FUNCTION_BLOCK FB_Regelschuif_AFO IMPLEMENTS ITF_Regelschuif
VAR
	tagName : STRING;
	outputOpen : ITF_Schuif_DigOutOpen_AFO;
	outputClose : ITF_Schuif_DigOutClose_AFO;
	inputPosition : ITF_Schuif_AnaIn_AFO;

	currentMode : E_Bedrijfstoestand := E_Bedrijfstoestand.off;
	currentState : E_RegelschuifState := E_RegelschuifState.standby;
	expectedState : E_RegelschuifState := E_RegelschuifState.standby;
	
	feedbackPosition : SINT;
	
	timeOut : TON;
	errorTrigger : R_TRIG;
	positie : SINT;
	secondTimerRun : BOOL;
	secondTimerTrigger : R_TRIG;
	
	timerrunt: BOOL:=1;
	waitExtraMinute: BOOL;
	minuteTimer : TON;
	doubleMinuteTimer : TON;
	secondTimer : TON;
	
	veranderingsMargeError : SINT := 3;
	OldPosition: SINT;
	regelschuifMargin: SINT := 3;
END_VAR

// Als de mode is uit dan worden de outputs false geset 
IF currentMode = E_Bedrijfstoestand.off THEN
	outputOpen.set(FALSE);
	outputClose.set(FALSE);
END_IF

// De feedback positie staat hiet zodat we de waardes kunnen veranderen
feedbackPosition := inputPosition.get();
ActueelPosition := inputPosition.get();

// Dit is de timer om te checken of er een error moet zijn 
timeOut(IN :=(StateRegelSchuif <> E_RegelschuifState.standby) AND NOT timeOut.Q, PT := T#30S);
errorTrigger(CLK := timeOut.Q);

IF errorTrigger.Q THEN
	IF (ActueelPosition < (OldPosition + veranderingsMargeError)) AND StateRegelSchuif = E_RegelschuifState.opening THEN
		StateRegelSchuif := E_RegelschuifState.error;
		main.alarms.append(tag := tagName, msg := 'Schuifstoring gedetecteerd, te langzaam openen');
	END_IF
	IF (ActueelPosition > (OldPosition - veranderingsMargeError)) AND StateRegelSchuif = E_RegelschuifState.closing THEN
		StateRegelSchuif := E_RegelschuifState.error;
		main.alarms.append(tag := tagName, msg := 'Schuifstoring gedetecteerd, te langzaam sluiten');
	END_IF
	IF StateRegelSchuif = E_RegelschuifState.error AND (ActueelPosition > (OldPosition + veranderingsMargeError)) THEN
		StateRegelSchuif := E_RegelschuifState.opening;
		ELSIF StateRegelSchuif = E_RegelschuifState.error AND (ActueelPosition < (OldPosition - veranderingsMargeError)) THEN
			StateRegelSchuif := E_RegelschuifState.closing;
	END_IF
	OldPosition := ActueelPosition;
END_IF

expectedState := StateRegelSchuif;

PROPERTY ActueelPosition : SINT
GET
ActueelPosition := feedbackPosition;
END_GET
SET
feedbackPosition := ActueelPosition;
END_SET
END_PROPERTY

//FB_Init is always available implicitly and it is used primarily for initialization.
//The return value is not evaluated. For a specific influence, you can also declare the
//methods explicitly and provide additional code there with the standard initialization
//code. You can evaluate the return value.
METHOD FB_Init: BOOL
VAR_INPUT
    bInitRetains: BOOL; // TRUE: the retain variables are initialized (reset warm / reset cold)
    bInCopyCode: BOOL;  // TRUE: the instance will be copied to the copy code afterward (online change)   
	tag : STRING;
	DigOutOpening : ITF_Schuif_DigOutOpen_AFO;
	DigOutClosing : ITF_Schuif_DigOutClose_AFO;
	AnaInPosition : ITF_Schuif_AnaIn_AFO;
END_VAR
tagname := tag;
outputOpen := DigOutOpening;
outputClose := DigOutClosing;
inputPosition := AnaInPosition;
END_METHOD

METHOD RegelSchuifGoTo : SINT
VAR	
	checkPositions : BOOL;
	currentstatet: E_RegelschuifState;
	secondTriggerTrigger: BOOL;
END_VAR
VAR_INPUT
	regelschuifdoel : SINT;
END_VAR
minuteTimer(IN:= timerrunt,PT:= T#10S);
doubleMinuteTimer(IN:= waitExtraMinute,PT:= T#10S); // tweede timer om een extra minuut te wachten na pulse maar niet langer te wachten met scannen

// dit is zodat het gefaseerd gaat een pulse per sec sturen
secondTimer(IN:= secondTimerRun,PT:= T#2S); // pulse lengte langer ivm testen

IF currentMode = E_Bedrijfstoestand.off THEN
	regelschuifdoel := ActueelPosition;
END_IF

IF minuteTimer.Q THEN
	
	IF ActueelPosition >= (regelschuifdoel - regelschuifMargin) AND ActueelPosition <= (regelschuifdoel + regelschuifMargin) THEN // huidige positie is correct binnen marge
		StateRegelSchuif := E_RegelschuifState.standby;
		outputOpen.set(FALSE); // set outputs naar 0 als extra backup
		outputClose.set(FALSE);
	
	END_IF
	
	IF ActueelPosition > (regelschuifdoel + regelschuifMargin) AND waitExtraMinute = FALSE THEN // huidige positie is te hoog
		IF stateRegelschuif <> E_RegelschuifState.error THEN
			StateRegelSchuif := E_RegelschuifState.closing;
		END_IF
		// voor de pulse		
		outputOpen.set(FALSE);
		outputClose.set(TRUE);
		secondTimerRun := TRUE; // start pulse time
		waitExtraMinute := TRUE; // wacht een minuut extra als er een pulse is gestuurd
	END_IF

	IF ActueelPosition < (regelschuifdoel - regelschuifMargin) AND waitExtraMinute = FALSE THEN // huidige positie is te laag
		IF stateRegelschuif <> E_RegelschuifState.error THEN
			StateRegelSchuif := E_RegelschuifState.opening;
		END_IF
		// voor de pulse
		outputClose.set(FALSE);
		outputOpen.set(TRUE);
		secondTimerRun := TRUE; // start pulse time
		waitExtraMinute := TRUE;
	END_IF
	timerrunt := 0; // reset timer
ELSIF waitExtraMinute = FALSE OR doubleMinuteTimer.Q THEN 
	waitExtraMinute := FALSE;
	timerrunt := 1; //reser reset timer
END_IF

// pulse timer structuur
IF secondTimer.Q THEN
	outputClose.set(FALSE);
	outputOpen.set(FALSE);
	secondTimerRun := FALSE;
END_IF

positie := regelschuifdoel;
END_METHOD

PROPERTY StateRegelSchuif : E_RegelschuifState
GET
StateRegelschuif := currentState;
END_GET
SET
currentstate:= StateRegelSchuif;
END_SET
END_PROPERTY

END_FUNCTION_BLOCK

(* stored: Version 1.1.0.1, ProductVersion 3.1.4026.8
   POU FB_Regelschuif_AFO: Id {e3716e21-c926-4b53-b092-edc4b4bb1690}, SpecialFunc None
   Folder Methods: Id {19e33316-aa4d-4340-a18c-c48173f3eae7}
   Folder Properties: Id {e2e5e1b1-49a7-46d0-8daf-b77eea7842e6}
   Property ActueelPosition: Id {2d2a6d11-befa-4588-8131-86e3894c6457}
   Get Get: Id {fc7c4d48-73b9-47ec-8f27-7cd7b636e38c}
   Set Set: Id {9454e573-b814-4817-822e-cf1729db9dd6}
   Method FB_Init: Id {3a2e7ee9-0040-407c-9fdc-e034eb20bdea}
   Method RegelSchuifGoTo: Id {79c61f24-d77f-47a4-b036-2823abebfb78}
   Property StateRegelSchuif: Id {970eafd1-96ea-40c0-b909-2be329c20549}
   Get Get: Id {75d5413c-e9a2-4d07-852b-3149b8f38d87}
   Set Set: Id {c2a73e76-74c5-4c09-8b03-2178d70ef95f} *)
